TEXTLIST CommandType
  0 = 'DISABLE'
  1 = 'MOVE'
  2 = 'PAUSE'
  3 = 'INPUT'
  4 = 'OUTPUT'
  5 = 'VISION'
  6 = 'CNC'
  7 = 'VARSET'
  8 = 'LOGIC'
   = ''
END_TEXTLIST

(* stored: Version 1.1.0.1
   TextList CommandType: Id {d449e393-ee4a-415a-9faf-628cd9281f9a} *)
